FUNCTION_BLOCK Motor_Dosagem (* Composite Function Block Type *)
  (* Standard: 61499-2 *)
  (* Version 0.0, 1/22/2026, Schneider Electric, template *)
  PACKAGE Hidryco.HidrycoLib;
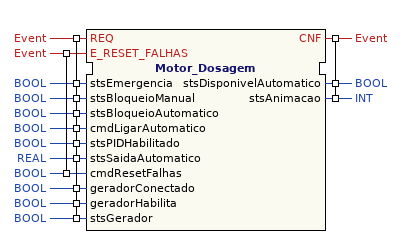
  EVENT_INPUT
    REQ WITH stsBloqueioManual, stsBloqueioAutomatico, cmdLigarAutomatico, stsPIDHabilitado, stsSaidaAutomatico, geradorConectado, geradorHabilita, stsGerador, stsEmergencia;
    E_RESET_FALHAS WITH cmdResetFalhas;
  END_EVENT
  EVENT_OUTPUT
    CNF WITH stsDisponivelAutomatico, stsAnimacao;
  END_EVENT
  VAR_INPUT
    stsEmergencia : BOOL;
    stsBloqueioManual : BOOL;
    stsBloqueioAutomatico : BOOL;
    cmdLigarAutomatico : BOOL;
    stsPIDHabilitado : BOOL;
    stsSaidaAutomatico : REAL;
    cmdResetFalhas : BOOL;
    geradorConectado : BOOL;
    geradorHabilita : BOOL;
    stsGerador : BOOL;
  END_VAR
  VAR_OUTPUT
    stsDisponivelAutomatico : BOOL;
    stsAnimacao : INT;
  END_VAR
  (* 0 - INITIALIZATION *)
  (* 1 - FUNCTIONAL INPUT INTERFACE *)
  (* 6 - OT-IT INTERFACE *)
  (* 2 - FUNCTIONAL OUTPUT INTERFACE *)
  (* 3 - FIELD INTERFACE *)
  (* 4 - CHILDREN *)
  (* 5 - LOGICS *)
  (* 5.B - OPERATION MODE MANAGEMENT *)
  (* 5.C - INTERLOCKS MANAGEMENT *)
  (* 5.A - FUNCTIONAL BEHAVIORS *)
  (* Verificar se precisa gravar a unidade *)
  FBS
    IThis : Motor_Dosagem_HMI(QI := TRUE);
    SYMLINKMULTIVARDST1 : SYMLINKMULTIVARDST_16501039F25307793(QI := TRUE, NAME1 := '$${PATH}stsLocal', NAME2 := '$${PATH}stsRemoto', NAME3 := '$${PATH}stsLigado', NAME4 := '$${PATH}stsFalha', NAME5 := '$${PATH}stsFalhaComunicacao', NAME6 := '$${PATH}stsFluxoInstantaneo', NAME7 := '$${PATH}stsProtecaoTermica'); {SET_ATTRIBUTE(Configuration.GenericFBType.InterfaceParams, Runtime.System#I:=7;VALUE${I$}:BOOL,BOOL,BOOL,BOOL,BOOL,REAL,BOOL)}
    SYMLINKMULTIVARSRC1 : SYMLINKMULTIVARSRC_804524063F215924(QI := TRUE, NAME1 := '$${PATH}cmdAcionamento', NAME2 := '$${PATH}stpSaida', NAME3 := '$${PATH}cmdReset'); {SET_ATTRIBUTE(Configuration.GenericFBType.InterfaceParams, Runtime.System#I:=3;VALUE${I$}:BOOL,REAL,BOOL)}
    plcStart1 : plcStart(Prio := 10);
  END_FBS
  EVENT_CONNECTIONS
    plcStart1.FIRST_INIT TO IThis.77A2F60CB33ACCE3;
    plcStart1.REDO_INIT TO IThis.77A2F60CB33ACCE3;
    SYMLINKMULTIVARDST1.CNF TO IThis.3E1D0BBAE7B97111;
    IThis.636E0523AE14AA92 TO IThis.3E1D0BBAE7B97111;
    IThis.E95E96A346CBF4D4 TO IThis.3E1D0BBAE7B97111;
    IThis.8988C31EE2188F23 TO IThis.885DC47239123EB9;
    IThis.8988C31EE2188F23 TO SYMLINKMULTIVARDST1.INIT;
    SYMLINKMULTIVARDST1.INITO TO SYMLINKMULTIVARSRC1.INIT;
    SYMLINKMULTIVARSRC1.INITO TO plcStart1.ACK_FIRST;
    E_RESET_FALHAS TO SYMLINKMULTIVARSRC1.REQ;
  END_CONNECTIONS
  DATA_CONNECTIONS
    SYMLINKMULTIVARDST1.VALUE2 TO IThis.841BF87C17BC0349;
    SYMLINKMULTIVARDST1.VALUE5 TO IThis.B8C930269FBFC965;
    SYMLINKMULTIVARDST1.VALUE6 TO IThis.E981264F18CB1FBA;
    IThis.3B54B4F232F61934 TO IThis.F2C3D7B089DF9B40;
    IThis.89F4F7CACE4761CD TO IThis.68C5779237D4A698;
    SYMLINKMULTIVARDST1.VALUE7 TO IThis.9599BF1F5A2F9D9B;
    SYMLINKMULTIVARDST1.VALUE3 TO IThis.8119E32988BA6026;
    cmdResetFalhas TO SYMLINKMULTIVARSRC1.VALUE3;
  END_CONNECTIONS
END_FUNCTION_BLOCK
